PROGRAM MAIN
VAR
	input1: BOOL;
	output1:BOOL;
	counter : int;
END_VAR

counter := counter +1;
light();

END_PROGRAM

(* stored: Version 1.1.0.1, ProductVersion 3.1.4024.12
   POU MAIN: Id {05dceb2c-0d53-456d-b815-0e85d7a4d0aa}, SpecialFunc None *)
